// TwinCAT 3 PLC project Untitled1
// ProgramVersion: 3.1.4026.20
// libraries:
//   Tc2_Standard, * (Beckhoff Automation GmbH)
//   Tc2_System, * (Beckhoff Automation GmbH)
// project tree:
//   / PlcTask.TcTTO, PlcTaskFast.TcTTO
//   POUs/ MAIN.TcPOU, MAINFast.TcPOU
// real-time tasks:
//   TASK PlcTask: cycle T#10ms, priority 20, ADS port 350
//   TASK PlcTaskFast: cycle T#5ms, priority 21, ADS port 351

CONFIGURATION Untitled1
    RESOURCE PLC ON TwinCAT3
        TASK PlcTask(INTERVAL := T#10ms, PRIORITY := 20);
        TASK PlcTaskFast(INTERVAL := T#5ms, PRIORITY := 21);
        PROGRAM MAIN WITH PlcTask : MAIN;
        PROGRAM MAINFast WITH PlcTaskFast : MAINFast;
    END_RESOURCE
END_CONFIGURATION

// ---- POUs/MAIN.TcPOU
PROGRAM MAIN
VAR
	test : BOOL;
END_VAR

test := NOT test;

END_PROGRAM

// ---- POUs/MAINFast.TcPOU
PROGRAM MAINFast
VAR
	test : BOOL;
END_VAR

test := NOT test;

END_PROGRAM
